// TwinCAT 3 PLC project RpcClient
// ProgramVersion: 3.1.4024.0
// libraries:
//   rplc, * (tchaxx)
//   Tc2_Standard, * (Beckhoff Automation GmbH)
//   Tc2_System, * (Beckhoff Automation GmbH)
//   Tc3_Module, * (Beckhoff Automation GmbH)
// project tree:
//   / PlcTask.TcTTO
//   POUs/ FB_Subscriber.TcPOU, MAIN.TcPOU

CONFIGURATION RpcClient
    RESOURCE PLC ON TwinCAT3
        TASK PlcTask(INTERVAL := T#10ms, PRIORITY := 22);
        PROGRAM MAIN WITH PlcTask : MAIN;
    END_RESOURCE
END_CONFIGURATION

// ---- POUs/MAIN.TcPOU
PROGRAM MAIN
VAR
	fbRpc		: tchaxx.FB_RPC(sAmsNetId:= tchaxx.GCL.cLocalAmsNetId, nAmsPort:= 852, sInstancePath:= 'MAIN.fbRpcServer', sSymbol:= 'Greet');
	
	// Arguments and RetVal
	sArg  : T_MaxString := _AppInfo.AppName;
	nLen  : INT;
	stLibVersion : ST_LibVersion := Tc3_Module.Global_Version.stLibVersion_Tc3_Module;
	sRetVal : T_MaxString;
	stRetVal : ST_AdsStatus;
	
	// PubSub example
	fbSubscriber1	:	FB_Subscriber(sInstancePath:= 'MAIN.fbSubscriber1');
	fbSubscriber2	:	FB_Subscriber(sInstancePath:= 'MAIN.fbSubscriber2');
END_VAR


stRetVal := fbRpc.VarInput(sArg)
                 .VarOutput(nLen)
                 .VarInOut(stLibVersion)
                 .ReturnValue(sRetVal)
                 .Invoke();
				 
fbSubscriber1();
fbSubscriber2();

END_PROGRAM

// ---- POUs/FB_Subscriber.TcPOU
FUNCTION_BLOCK FINAL FB_Subscriber
VAR_INPUT
END_VAR
VAR_OUTPUT
END_VAR
VAR
	fbRpcPublisherSubscribe 	: tchaxx.FB_RPC(sAmsNetId:= tchaxx.GCL.cLocalAmsNetId, nAmsPort:= 852, sInstancePath:= 'MAIN.fbPublisher', sSymbol:= 'Subscribe');
	fbRpcPublisherUnsubscribe 	: tchaxx.FB_RPC(sAmsNetId:= tchaxx.GCL.cLocalAmsNetId, nAmsPort:= 852, sInstancePath:= 'MAIN.fbPublisher', sSymbol:= 'Unsubscribe');
	sInstancePath			: STRING;
	sSymbolCallback			: STRING := 'PublisherEventCallback';
	nHandle					: UDINT;
	nValuePublished			: UDINT;
	bSubscribe				: BOOL := TRUE;
	bUnsubscribe			: BOOL := FALSE;
	bSubscribed				: BOOL := FALSE;
	stAdsStatus				: tchaxx.ST_AdsStatus;
END_VAR

VAR_TEMP
	sAmsNetId	: T_AmsNetID := tchaxx.GCL.cLocalAmsNetId;
	hr		 	: HRESULT;
END_VAR

IF NOT bSubscribed AND bSubscribe THEN
	stAdsStatus := fbRpcPublisherSubscribe.VarInput(anyArg:= sAmsNetId)
					.VarInput(anyArg:= _AppInfo.AdsPort)
					.VarInput(anyArg:= sInstancePath)
					.VarInput(anyArg:= sSymbolCallback)
					.VarOutput(anyArg:= nHandle)
					.ReturnValue(anyRetVal:= hr)
					.Invoke();
					
	bSubscribed := NOT stAdsStatus.bBusy AND NOT stAdsStatus.bError;
	IF bSubscribed THEN
		bSubscribe := FALSE;
	END_IF
END_IF;
				
IF bSubscribed AND bUnsubscribe THEN
	stAdsStatus := fbRpcPublisherUnsubscribe.VarInput(anyArg:= nHandle).ReturnValue(anyRetVal:= hr).Invoke();
	IF NOT stAdsStatus.bBusy AND NOT stAdsStatus.bError THEN
		bSubscribed := FALSE;
		bUnsubscribe := FALSE;
	END_IF
END_IF

METHOD FB_init : BOOL
VAR_INPUT
	bInitRetains : BOOL; // if TRUE, the retain variables are initialized (warm start / cold start)
	bInCopyCode : BOOL;  // if TRUE, the instance afterwards gets moved into the copy code (online change)
	sInstancePath : STRING;
END_VAR
THIS^.sInstancePath := sInstancePath;
END_METHOD

{attribute 'TcRpcEnable'}
METHOD PRIVATE PublisherEventCallback
VAR_INPUT
	nValue	: UDINT;
END_VAR

nValuePublished := nValue;
END_METHOD

END_FUNCTION_BLOCK
